	FUNCTION_BLOCK FB 116
	TITLE =G016M CCOMPRESSED AIR PRESSURE STEEP 5 - 8
	//COPYRIGHT:    (C) 2009  BUHLER AG, CH-9240 UZWIL, SWITZERLAND
	//
	//PRODUCT:      WinCoS_BIW01_09
	//
	//TITLE:        CCOMPRESSED AIR PRESSURE STEEP 5 - 8
	//                Machine group control
	//                Maschinengruppensteuerung
	//
	//--------------------------------------------------------------------------------
	//
	//IDENT:        AUTHOR:             DEPT:                              DATE:
	//
	//P01_FB116.1.0 K.Renz              CSB41                              13.Jan.2010
	//             1st Release
	//
	//--------------------------------------------------------------------------------
	//
	//PURPOSE:
	//
	//MANUAL :
	//
	//RESTRICTIONS:
	//
	//--------------------------------------------------------------------------------
	AUTHOR  : KR
	FAMILY  : USW
	VERSION : 9.9


	VAR
	  Gr       : FB10;	//Standard interface to group
	  InOutValue1    : DINT; //Data for user
	  InOutValue2    : DINT; //Data for user
	  OutWayConflict : BOOL;	//Data for user
	  OutSelectionOk : BOOL;	//Data for user
	  CmdNewValue : BOOL;	//Data for user
	  CmdNewJob   : BOOL;	//Data for user
	  OutCodeOK   : BOOL;	//Data for user
	  InEndOfJob  : BOOL ;	//Data for user
	  staWayOk      : BOOL ;	//Data for user
	  EdgeStartRelease : BOOL ;	//Data for user
	  USW8  : BOOL;	//Data for user
	  USW9 : BOOL;	//Data for user
	  USW10: BOOL;	//Data for user
	  USW11: BOOL;	//Data for user
	  USW12: BOOL;	//Data for user
	  USW13: BOOL;	//Data for user
	  USW14: BOOL;	//Data for user
	  USW15: BOOL;	//Data for user
	     #A_1152_MXZ11 : FB12;   // Motor
	END_VAR
	VAR_TEMP
	   tmpEnable		: BOOL;
	   tmpFlag  		: BOOL;
	   tmpCmdNext		: BOOL;
	   tmpLocal  		: BOOL;
	   tmpAspOk  		: BOOL;
	   tmpHWStop 		: BOOL;
	   tmpInstanzDBNo       : INT ;
	END_VAR
	BEGIN
	NETWORK
	TITLE =
	NETWORK
	TITLE =Read command from group control
	//Parameter
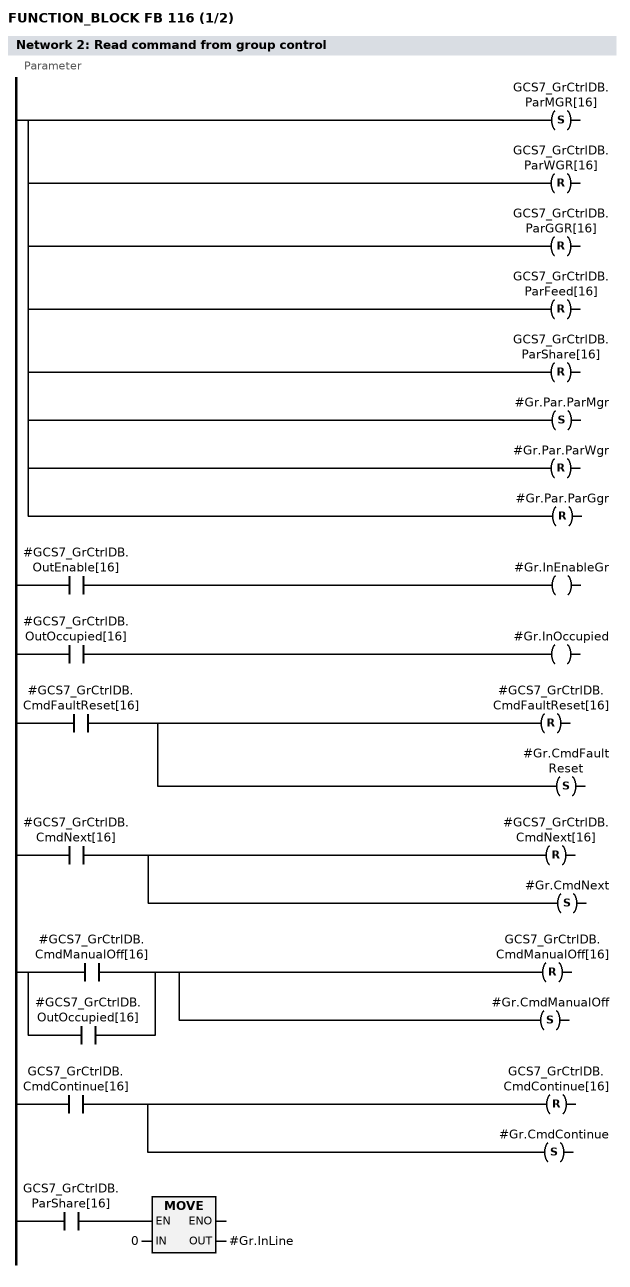
	      SET;
	      S   GCS7_GrCtrlDB.ParMGR[16];
	      R   GCS7_GrCtrlDB.ParWGR[16];
	      R   GCS7_GrCtrlDB.ParGGR[16];
	      R   GCS7_GrCtrlDB.ParFeed[16];
	      R   GCS7_GrCtrlDB.ParShare[16];
	      S   #Gr.Par.ParMgr;
	      R   #Gr.Par.ParWgr;
	      R   #Gr.Par.ParGgr;
	//Command
	      U   #GCS7_GrCtrlDB.OutEnable[16];
	      =   #Gr.InEnableGr;
	      U   #GCS7_GrCtrlDB.OutOccupied[16];
	      =   #Gr.InOccupied;
	      U   #GCS7_GrCtrlDB.CmdFaultReset[16];
	      R   #GCS7_GrCtrlDB.CmdFaultReset[16];
	      S   #Gr.CmdFaultReset;
	      U  #GCS7_GrCtrlDB.CmdNext[16];
	      R   #GCS7_GrCtrlDB.CmdNext[16];
	      S   #Gr.CmdNext;
	      U   #GCS7_GrCtrlDB.CmdManualOff[16];
	      O   #GCS7_GrCtrlDB.OutOccupied[16];
	      R   GCS7_GrCtrlDB.CmdManualOff[16];
	      S   #Gr.CmdManualOff;
	      U  GCS7_GrCtrlDB.CmdContinue[16];
	      R   GCS7_GrCtrlDB.CmdContinue[16];
	      S   #Gr.CmdContinue;
	//Init Line Number
	      U   GCS7_GrCtrlDB.ParShare[16];
	      SPBN WE00;
	      L     0;
	      T     #Gr.InLine;
	WE00: NOP   0;
	NETWORK
	TITLE =Call Methode Control
	// 1. Handle Interface PCControl
	// 2. Prepare mode --> ModePassive,ModeActive,ModeIdling
	// 3. Reset global flags of the group
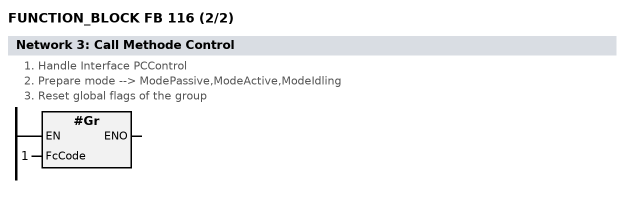
	      CALL #Gr (
	           FcCode                   := 1);
	NETWORK
	TITLE =Restart Idling Time
		L  #Gr.Par.ParIdling;
		L  2;
		>=I;
		SPB IdTm;
		T  #Gr.Par.ParIdling;
	IdTm:   NOP 0;
	      CLR;
	      S    #Gr.CmdRestartIdling;
	NETWORK
	TITLE =Prepare global flags
	NETWORK
	TITLE =Set Pattern (Target position)
	NETWORK
	TITLE =Interlocking WayOk
	//
	NETWORK
	TITLE =Interlocking Autostart
		CLR;
		R   #Gr.OutAutostart;
	NETWORK
	TITLE =Interlocking Enable
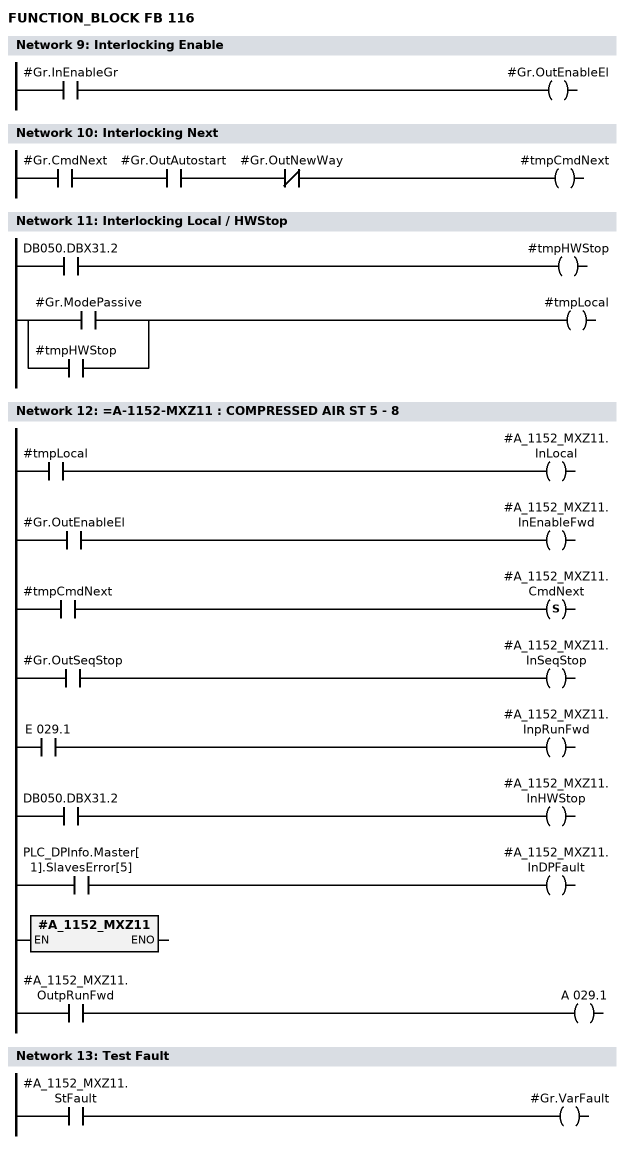
	      U     #Gr.InEnableGr;
	      =     #Gr.OutEnableEl;

	NETWORK
	TITLE =Interlocking Next
	      U     #Gr.CmdNext;
	      U     #Gr.OutAutostart;
	      UN    #Gr.OutNewWay;
	      =    #tmpCmdNext;

	NETWORK
	TITLE =Interlocking Local / HWStop
	      U    DB050.DBX31.2;
	      =    #tmpHWStop;

	      U    #Gr.ModePassive;
	      O    #tmpHWStop;
	      =    #tmpLocal;

	NETWORK
	TITLE ==A-1152-MXZ11 : COMPRESSED AIR ST 5 - 8
	NOP 0;
	//-InLocal---
	      U     #tmpLocal;
	      =     #A_1152_MXZ11.InLocal;
	//
	//-Interlocking---
	      U     #Gr.OutEnableEl;
	      =     #A_1152_MXZ11.InEnableFwd;
	//
	      U    #tmpCmdNext;
	      S     #A_1152_MXZ11.CmdNext;
	//
	      U     #Gr.OutSeqStop;
	      =     #A_1152_MXZ11.InSeqStop;
	//
	//-Read inputs---
	      U     E 029.1;
	      =     #A_1152_MXZ11.InpRunFwd;
	      U   DB050.DBX31.2;
	      =     #A_1152_MXZ11.InHWStop;
	       U     PLC_DPInfo.Master[1].SlavesError[5];
	       =       #A_1152_MXZ11.InDPFault;
	//
	//-Set Parameters---
	//
	//-Call object control---
	      CALL  #A_1152_MXZ11;
	//
	//-Write outputs---
	      U     #A_1152_MXZ11.OutpRunFwd;
	      =     A 029.1;
	NETWORK
	TITLE =Test Fault
	      U     #A_1152_MXZ11.StFault;
	      =     #Gr.VarFault;
	NETWORK
	TITLE =Test Warning
	      CLR;
	      =     #Gr.OutWarning;
	NETWORK
	TITLE =Test Stopped
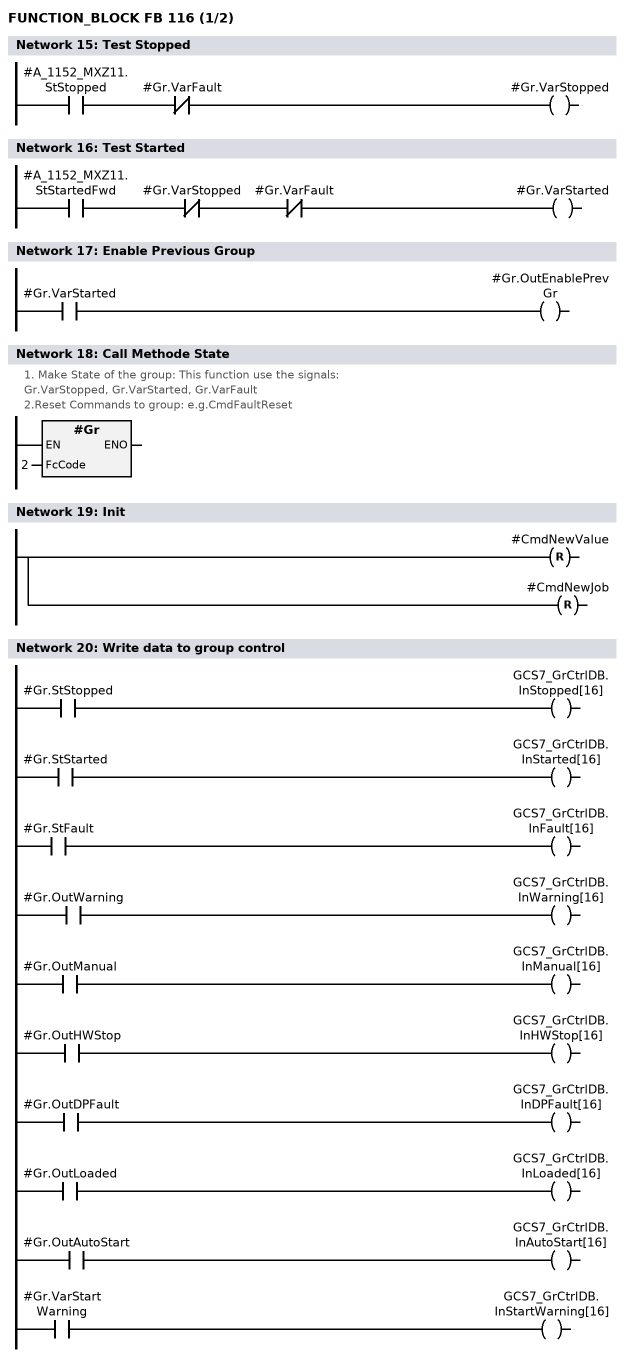
	      U     #A_1152_MXZ11.StStopped;
	      UN   #Gr.VarFault;
	      =     #Gr.VarStopped;
	NETWORK
	TITLE =Test Started
	      U     #A_1152_MXZ11.StStartedFwd;
	      UN  #Gr.VarStopped;
	      UN  #Gr.VarFault;
	      =     #Gr.VarStarted;
	NETWORK
	TITLE =Enable Previous Group
	      U    #Gr.VarStarted;
	      =     #Gr.OutEnablePrevGr;
	NETWORK
	TITLE =Call Methode State
	//1. Make State of the group: This function use the signals:
	//        Gr.VarStopped, Gr.VarStarted, Gr.VarFault
	//2.Reset Commands to group: e.g.CmdFaultReset
	      CALL #Gr (
	           FcCode                   := 2);
	NETWORK
	TITLE =Init
	      SET;
	      R    #CmdNewValue;
	      R    #CmdNewJob;
	NETWORK
	TITLE =Write data to group control
	      U   #Gr.StStopped;
	      =   GCS7_GrCtrlDB.InStopped[16];
	      U   #Gr.StStarted;
	      =   GCS7_GrCtrlDB.InStarted[16];
	      U   #Gr.StFault;
	      =   GCS7_GrCtrlDB.InFault[16];
	      U   #Gr.OutWarning;
	      =   GCS7_GrCtrlDB.InWarning[16];
	      U   #Gr.OutManual;
	      =   GCS7_GrCtrlDB.InManual[16];
	      U   #Gr.OutHWStop;
	      =   GCS7_GrCtrlDB.InHWStop[16];
	      U   #Gr.OutDPFault;
	      =   GCS7_GrCtrlDB.InDPFault[16];
	      U   #Gr.OutLoaded;
	      =   GCS7_GrCtrlDB.InLoaded[16];
	      U   #Gr.OutAutoStart;
	      =   GCS7_GrCtrlDB.InAutoStart[16];
	      U   #Gr.VarStartWarning;
	      =   GCS7_GrCtrlDB.InStartWarning[16];
	NETWORK
	TITLE =End of block
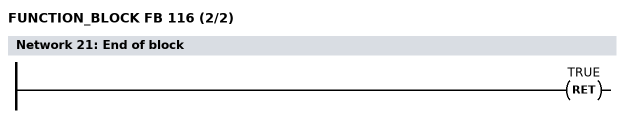

	BE

	END_FUNCTION_BLOCK
